INTERFACE I_LightTowerComponent

// Sets the component state to TRUE.
METHOD Activate
VAR_INPUT
END_VAR
END_METHOD

// Sets the component state to FALSE.
METHOD Deactivate
VAR_INPUT
END_VAR
END_METHOD

METHOD PulseWithInterval
VAR_INPUT
	DurationOn	: TIME;
	DurationOff	: TIME;
END_VAR
END_METHOD

END_INTERFACE

(* stored: Version 1.1.0.1, ProductVersion 3.1.4024.14
   Itf I_LightTowerComponent: Id {bc41dd1f-d349-051a-1eec-8006b1e366d0}
   Method Activate: Id {1ad27726-45d6-07ee-2f42-79a634ec1abf}
   Method Deactivate: Id {8a75ec4a-781b-011a-0a50-d3a598bef27a}
   Method PulseWithInterval: Id {4e473a09-f3d1-049e-0a52-d0f47ca47dd1} *)
